# EPICS substitutions: ek9000App/Db/EL3061.substitutions
file EL3061.template
{       pattern
        {
                TERMINAL,

        }
        {
        }
}
